{attribute addProperty BoxType "AX5101-0000-0005-0005"}
{attribute addProperty Id "AT_xAT %I*AT_x_029F01154860MDTAT %Q*MDT_47A878CF4860WcStateAT %I*WcState_98A4DF7520.250InfoDataAT %I*InfoData_AEB17F4D152190"}
{attribute addProperty CRC "245682833"}
{attribute addProperty SizeInBites "250"}
{attribute addProperty SizeInBytes "31.25"}
TYPE AX5101_47F5CC47 :
STRUCT
	{attribute addProperty Name "AT_x"}
	AT_x : AT_x_029F0115;
	{attribute addProperty Name "MDT"}
	MDT : MDT_47A878CF;
	{attribute addProperty Name "WcState"}
	WcState : WcState_98A4DF75;
	{attribute addProperty Name "InfoData"}
	InfoData : InfoData_AEB17F4D;
END_STRUCT
END_TYPE

(* stored: Version 1.2.0.0, ProductVersion 3.1.4024.9
   DUT AX5101_47F5CC47: Id {257e864a-c253-43f5-a714-25cd00e2948b} *)
